FUNCTION_BLOCK FB_buffer
VAR_INPUT
END_VAR
VAR_OUTPUT
END_VAR
VAR

	fb_rollers		: ARRAY[0..iHas_rollers] OF FB_roller;
	sensor_start	: ARRAY[0..1] OF FB_DigitalInput;//sensor at the beginning of roller[0]
	EDM_24v	: BOOL;//edm_24v
	EDM_sto	: BOOL;//edm_sto
	xError	: BOOL;
	
	i	: INT;
	event				: ST_EVENT;
	rt_error			: R_TRIG;
END_VAR
VAR CONSTANT
	iHas_rollers	: INT:=3;
	sComponent_name			: STRING := 'fb_buffer';
END_VAR

M_mapping();
event.sTime	:= MAIN.Temp_str;
event.sComponent_name	:= sComponent_name;
xError	:= fb_rollers[0].xError OR fb_rollers[1].xError OR fb_rollers[2].xError  OR fb_rollers[3].xError;

METHOD M_agingTest : BOOL
VAR_INPUT
END_VAR
FOR i:=0 TO iHas_rollers DO
	fb_rollers[i].M_agingTest();
END_FOR
END_METHOD

METHOD M_init : BOOL
VAR_INPUT
END_VAR
VAR
	i: INT;
END_VAR
M_init	:= FALSE;

FOR i:=0 TO iHas_rollers DO
	fb_rollers[i].M_init();
END_FOR
xError	:= FALSE;
M_init	:= TRUE;
END_METHOD

METHOD M_mapping : BOOL
VAR_INPUT
END_VAR

//todo:reconfig dios
/////////////////////////////////////digital input////////////////////////////////////////

fb_rollers[0].roller.err			:= G_IO.arDI[1].Ch[0];
fb_rollers[1].roller.err			:= G_IO.arDI[1].Ch[1];
fb_rollers[1].roller.sensor(D:= G_IO.arDI[1].Ch[2],on_ms:=100,off_ms:=100);
fb_rollers[2].roller.sensor(D:= G_IO.arDI[1].Ch[3],on_ms:=100,off_ms:=100);
fb_rollers[2].roller.err			:= G_IO.arDI[1].Ch[4];
fb_rollers[3].roller.err			:= G_IO.arDI[1].Ch[5];
fb_rollers[3].roller.sensor(D:= G_IO.arDI[1].Ch[6],on_ms:=100,off_ms:=100);
fb_rollers[3].sensor_mute(D:= G_IO.arDI[1].Ch[7],on_ms:=10,off_ms:=100);
EDM_24v								:= G_IO.arDI[1].Ch[11];
EDM_sto								:= G_IO.arDI[1].Ch[12];
sensor_start[0](D:= G_IO.arDI[1].Ch[13],on_ms:=100,off_ms:=100);
sensor_start[1](D:= G_IO.arDI[1].Ch[15],on_ms:=100,off_ms:=100);
fb_rollers[0].roller.sensor(D:= G_IO.arDI[1].Ch[14],on_ms:=100,off_ms:=100);

/////////////////////////////////////digital output////////////////////////////////////////
G_IO.arDO[1].Ch[0]	:= fb_rollers[2].roller.forward;
G_IO.arDO[1].Ch[1]	:= fb_rollers[2].roller.backward;
G_IO.arDO[1].Ch[2]	:= fb_rollers[0].roller.forward;
G_IO.arDO[1].Ch[3]	:= fb_rollers[0].roller.backward;
G_IO.arDO[1].Ch[4]	:= fb_rollers[1].roller.forward;
G_IO.arDO[1].Ch[5]	:= fb_rollers[1].roller.backward;
G_IO.arDO[1].Ch[6]	:= fb_rollers[3].roller.forward;
G_IO.arDO[1].Ch[7]	:= fb_rollers[3].roller.backward;



/////////////////////////////////////fb rollers////////////////////////////////////////

FOR i:=0 TO iHas_rollers DO
	fb_rollers[i].M_mapping(i);
END_FOR
END_METHOD

METHOD M_reset : BOOL
VAR_INPUT
END_VAR

VAR
	i: INT;
END_VAR
M_reset	:= FALSE;

FOR i:=0 TO iHas_rollers DO
	IF fb_rollers[i].M_reset() THEN
		CONTINUE;
	END_IF
END_FOR

M_reset	:= TRUE;
END_METHOD

METHOD M_run : BOOL
VAR_INPUT
END_VAR
M_run	:= FALSE;
IF sensor_start[0].Q OR sensor_start[1].Q THEN
	fb_rollers[0].pre_tote_status := ToteStatus.READY;
ELSE
	fb_rollers[0].pre_tote_status := ToteStatus.EMPTY;
END_IF
fb_rollers[0](	id_roller := 0,
				next_tote_status := fb_rollers[1].current_tote_status);
fb_rollers[1](	id_roller := 1,
				pre_tote_status := fb_rollers[0].current_tote_status,
				next_tote_status := fb_rollers[2].current_tote_status);
fb_rollers[2](	id_roller := 2,
				pre_tote_status := fb_rollers[1].current_tote_status,
				next_tote_status := fb_rollers[3].current_tote_status);
fb_rollers[3](	id_roller := 3,
				pre_tote_status := fb_rollers[2].current_tote_status,
				next_tote_status := GVL.fb_loading.current_tote_status);
END_METHOD

METHOD M_runStart : BOOL
VAR_INPUT
END_VAR
VAR
	pSt_mcAxis	:POINTER TO ST_MotionAxis_MC;
END_VAR
M_runStart	:= FALSE;
pSt_mcAxis	:= ADR(fb_rollers[3].st_mcAxis);
pSt_mcAxis^.mcPower.Enable	:= TRUE;
IF pSt_mcAxis^.mcReadStatus.StandStill THEN
	M_runStart	:= TRUE;
END_IF
END_METHOD

METHOD M_safetyEvent : BOOL
VAR_INPUT
END_VAR
FOR i:=0 TO iHas_rollers DO
	fb_rollers[i].M_safetyEvent();
END_FOR
END_METHOD

END_FUNCTION_BLOCK

(* stored: Version 1.1.0.1, ProductVersion 3.1.4024.12
   POU FB_buffer: Id {df2ad2d1-8c07-4422-b79c-40aa917c064c}, SpecialFunc None
   Method M_agingTest: Id {1df7ec77-4153-4cd2-b633-bc1e438b8593}
   Method M_init: Id {32549cd6-4604-40a8-a88c-7b7c334ab582}
   Method M_mapping: Id {1a6da0bb-d604-4476-be71-0afdb8d7c5db}
   Method M_reset: Id {0155cc58-4f6d-443b-9601-ef576d9314eb}
   Method M_run: Id {2da5b0e5-7de5-409a-8737-9e1baf67abf8}
   Method M_runStart: Id {e71d628c-dfad-4383-9c73-20739fe7da03}
   Method M_safetyEvent: Id {672a5a87-b7ca-4286-9a78-13df69728b10} *)
